KUKA KRL program: ps_ltc_geo_x1.src, ps_ltc_geo_x1.dat

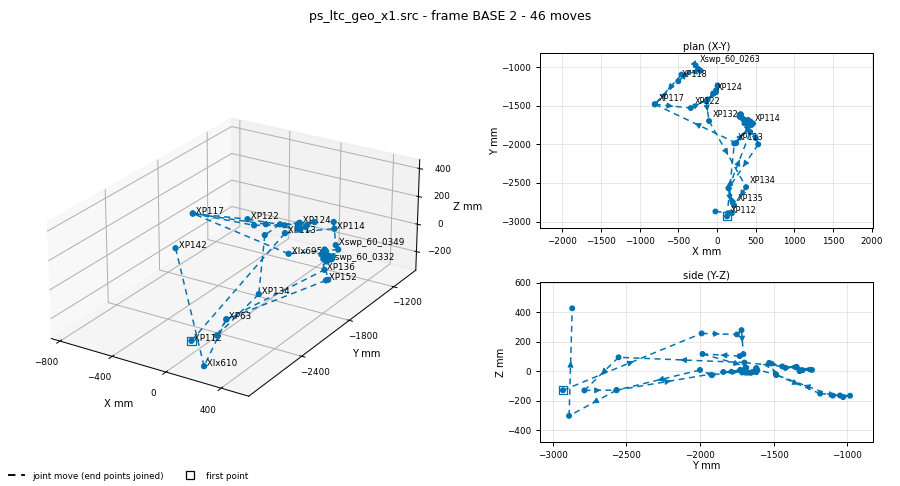
[picture p0: tool path of ps_ltc_geo_x1.src in frame BASE 2, 46 of 48 moves have a stored position in this frame; points joined in program order, loops and branches not executed]
--- ps_ltc_geo_x1.src ---
&ACCESS RVO2
&REL 17
&COMMENT Solda GUN X1 geometria
&PARAM DISKPATH = KRC:\R1\Program\SOLDA LTC
DEF ps_ltc_geo_x1( )
;FOLD INI
  ;FOLD BASISTECH INI
    GLOBAL INTERRUPT DECL 3 WHEN $STOPMESS==TRUE DO IR_STOPM ( )
    INTERRUPT ON 3
    BAS (#INITMOV,0 )
  ;ENDFOLD (BASISTECH INI)
;FOLD SPOTTECH INI
USERSPOT(#INIT)
;ENDFOLD (SPOTTECH INI)
;FOLD GRIPPERTECH INI
USER_GRP(0,DUMMY,DUMMY,GDEFAULT)
;ENDFOLD (GRIPPERTECH INI)
  ;FOLD USER INI
    ;Make your modifications here

  ;ENDFOLD (USER INI)
;ENDFOLD (INI)

; Caracterização dos meios de produção:
; Versão Atual:
; 08/06/2013 12:00 Name: P13.050-R1 CHANGES: Solda Geometria Accelo
; Gun X1 (F2 6640 0018 985)

chk_w1_wechs_ok ( )              ; CHECK X1

if MaxStandMenge (4) then
 MaxStandmengeErreicht (4)
endif

IF (NOT(GHOST())) THEN
if Elektrodenwechsel (4) then
 e_fraes1 ()
endif
ENDIF

;FOLD PTP P112 Vel=100 % PDAT114 Tool[1]:GUN X1 Base[2]:Accelo;%{PE}%R 8.2.20,%MKUKATPBASIS,%CMOVE,%VPTP,%P 1:PTP, 2:P112, 3:, 5:100, 7:PDAT114
$BWDSTART=FALSE
PDAT_ACT=PPDAT114
FDAT_ACT=FP112
BAS(#PTP_PARAMS,100)
PTP XP112
;ENDFOLD

;FOLD OUT 3339 'R1 solicita lib soldar geometria' State=TRUE ;%{PE}%R 8.2.20,%MKUKATPBASIS,%COUT,%VOUTX,%P 2:3339, 3:R1 solicita lib soldar geometria, 5:TRUE, 6:
$OUT[3339]=TRUE
;ENDFOLD
;FOLD WAIT FOR ( IN 3339 'Aguarda lib. Soldar geometria' );%{PE}%R 8.2.20,%MKUKATPBASIS,%CEXT_WAIT_FOR,%VEXT_WAIT_FOR,%P 2:, 4:, 5:$IN, 6:3339, 7:Aguarda lib. Soldar geometria, 9:
WAIT FOR  ( $IN[3339] )
;ENDFOLD
;FOLD OUT 3339 'R1 solicita lib soldar geometria' State=FALSE ;%{PE}%R 8.2.20,%MKUKATPBASIS,%COUT,%VOUTX,%P 2:3339, 3:R1 solicita lib soldar geometria, 5:FALSE, 6:
$OUT[3339]=FALSE
;ENDFOLD
;FOLD OUT 3348 'Fora area GEOBOX' State=FALSE ;%{PE}%R 8.2.20,%MKUKATPBASIS,%COUT,%VOUTX,%P 2:3348, 3:Fora area GEOBOX, 5:FALSE, 6:
$OUT[3348]=FALSE
;ENDFOLD

;FOLD Collision.Monitoring_3_On ;%{PE}%MKUKATPUSER
COLLSTOP( 3, 1 ) ;Interrupt-Controlled
;ENDFOLD
;FOLD Collision.Monitoring_AREA_1_On ;%{PE}%MKUKATPUSER
COLLSTOP( 7, 1 ) ;not Interrupt-Controlled
;ENDFOLD

;FOLD PTP P113 CONT Vel=100 % PDAT115 Tool[1]:GUN X1 Base[2]:Accelo;%{PE}%R 8.2.20,%MKUKATPBASIS,%CMOVE,%VPTP,%P 1:PTP, 2:P113, 3:C_DIS, 5:100, 7:PDAT115
$BWDSTART=FALSE
PDAT_ACT=PPDAT115
FDAT_ACT=FP113
BAS(#PTP_PARAMS,100)
PTP XP113 C_DIS
;ENDFOLD
;FOLD PTP P114 CONT Vel=100 % PDAT116 Tool[1]:GUN X1 Base[2]:Accelo;%{PE}%R 8.2.20,%MKUKATPBASIS,%CMOVE,%VPTP,%P 1:PTP, 2:P114, 3:C_DIS, 5:100, 7:PDAT116
$BWDSTART=FALSE
PDAT_ACT=PPDAT116
FDAT_ACT=FP114
BAS(#PTP_PARAMS,100)
PTP XP114 C_DIS
;ENDFOLD

;FOLD ; swp_60_0355;%{PE}%R 8.2.20,%MKUKATPBASIS,%CCOMMENT,%VNORMAL,%P 2:swp_60_0355
;ENDFOLD
;FOLD PTP swp_60_0355 P_OLP80 SPOT Gun=4 RETR CLS PGNO1=106 ACTIVE=1 Tool[1]:GUN X1 Base[2]:Accelo;%{PE}%R 8.2.2,%MKUKATPSPOT,%CSPOT,%VPTP,%P 1:PTP, 2:swp_60_0355, 3:, 5:100, 7:P_OLP80, 10:4, 12:#FIRST, 14:#CLO, 16:187, 18:1, 20:1, 22:0, 24:1, 25:S_OLP4
$BWDSTART=FALSE
PDAT_ACT=PP_OLP80
FDAT_ACT=Fswp_60_0355
BAS(#PTP_PARAMS,PP_OLP80.VEL)
S_ACT.GUN=4
S_ACT.PAIR=SDEFAULT.PAIR
S_ACT.RETR=#CLO
S_ACT.CLO_TM=1
S_ACT.PGNO1=106
S_ACT.PGNO2=SDEFAULT.PGNO2
S_ACT.PRESS1=SDEFAULT.PRESS1
S_ACT.PRESS2=SDEFAULT.PRESS2
S_READY=FALSE
PTP Xswp_60_0355
USERSPOT(#SPOT, S_ACT)
WAIT FOR S_READY
;ENDFOLD

;FOLD ; swp_60_0349;%{PE}%R 8.2.20,%MKUKATPBASIS,%CCOMMENT,%VNORMAL,%P 2:swp_60_0349
;ENDFOLD
;FOLD PTP swp_60_0349 P_OLP81 SPOT Gun=4 RETR OPN PGNO1=105 ACTIVE=1 Tool[1]:GUN X1 Base[2]:Accelo;%{PE}%R 8.2.2,%MKUKATPSPOT,%CSPOT,%VPTP,%P 1:PTP, 2:swp_60_0349, 3:, 5:100, 7:P_OLP81, 10:4, 12:#FIRST, 14:#OPN, 16:186, 18:1, 20:1, 22:0, 24:1, 25:S_OLP5
$BWDSTART=FALSE
PDAT_ACT=PP_OLP81
FDAT_ACT=Fswp_60_0349
BAS(#PTP_PARAMS,PP_OLP81.VEL)
S_ACT.GUN=4
S_ACT.PAIR=SDEFAULT.PAIR
S_ACT.RETR=#OPN
S_ACT.CLO_TM=1
S_ACT.PGNO1=105
S_ACT.PGNO2=SDEFAULT.PGNO2
S_ACT.PRESS1=SDEFAULT.PRESS1
S_ACT.PRESS2=SDEFAULT.PRESS2
S_READY=FALSE
PTP Xswp_60_0349
USERSPOT(#SPOT, S_ACT)
WAIT FOR S_READY
;ENDFOLD

;FOLD PTP P115 CONT Vel=100 % PDAT117 Tool[1]:GUN X1 Base[2]:Accelo;%{PE}%R 8.2.20,%MKUKATPBASIS,%CMOVE,%VPTP,%P 1:PTP, 2:P115, 3:C_DIS, 5:100, 7:PDAT117
$BWDSTART=FALSE
PDAT_ACT=PPDAT117
FDAT_ACT=FP115
BAS(#PTP_PARAMS,100)
PTP XP115 C_DIS
;ENDFOLD
;FOLD PTP lx695 Vel=100 % P_OLP82 Tool[1]:GUN X1 Base[2]:Accelo;%{PE}%R 8.2.20,%MKUKATPBASIS,%CMOVE,%VPTP,%P 1:PTP, 2:lx695, 3:, 5:100, 7:P_OLP82
$BWDSTART=FALSE
PDAT_ACT=PP_OLP82
FDAT_ACT=Flx695
BAS(#PTP_PARAMS,100)
PTP Xlx695
;ENDFOLD

;FOLD Collision.Monitoring_AREA_3_On ;%{PE}%MKUKATPUSER
COLLSTOP( 9, 1 ) ;not Interrupt-Controlled
;ENDFOLD

;FOLD PTP P117 CONT Vel=100 % PDAT119 Tool[1]:GUN X1 Base[2]:Accelo;%{PE}%R 8.2.20,%MKUKATPBASIS,%CMOVE,%VPTP,%P 1:PTP, 2:P117, 3:C_DIS, 5:100, 7:PDAT119
$BWDSTART=FALSE
PDAT_ACT=PPDAT119
FDAT_ACT=FP117
BAS(#PTP_PARAMS,100)
PTP XP117 C_DIS
;ENDFOLD
;FOLD PTP P118 CONT Vel=100 % PDAT120 Tool[1]:GUN X1 Base[2]:Accelo;%{PE}%R 8.2.20,%MKUKATPBASIS,%CMOVE,%VPTP,%P 1:PTP, 2:P118, 3:C_DIS, 5:100, 7:PDAT120
$BWDSTART=FALSE
PDAT_ACT=PPDAT120
FDAT_ACT=FP118
BAS(#PTP_PARAMS,100)
PTP XP118 C_DIS
;ENDFOLD

;FOLD ; swp_60_0263;%{PE}%R 8.2.20,%MKUKATPBASIS,%CCOMMENT,%VNORMAL,%P 2:swp_60_0263
;ENDFOLD
;FOLD PTP swp_60_0263 PDAT121 SPOT Gun=4 RETR CLS PGNO1=100 ACTIVE=1 Tool[1]:GUN X1 Base[2]:Accelo;%{PE}%R 8.2.2,%MKUKATPSPOT,%CSPOT,%VPTP,%P 1:PTP, 2:swp_60_0263, 3:, 5:100, 7:PDAT121, 10:4, 12:#FIRST, 14:#CLO, 16:181, 18:1, 20:0, 22:0, 24:1, 25:NORMAL
$BWDSTART=FALSE
PDAT_ACT=PPDAT121
FDAT_ACT=Fswp_60_0263
BAS(#PTP_PARAMS,PPDAT121.VEL)
S_ACT.GUN=4
S_ACT.PAIR=SDEFAULT.PAIR
S_ACT.RETR=#CLO
S_ACT.CLO_TM=1
S_ACT.PGNO1=100
S_ACT.PGNO2=SDEFAULT.PGNO2
S_ACT.PRESS1=SDEFAULT.PRESS1
S_ACT.PRESS2=SDEFAULT.PRESS2
S_READY=FALSE
PTP Xswp_60_0263
USERSPOT(#SPOT, S_ACT)
WAIT FOR S_READY
;ENDFOLD

;FOLD PTP P120 CONT Vel=100 % PDAT122 Tool[1]:GUN X1 Base[2]:Accelo;%{PE}%R 8.2.20,%MKUKATPBASIS,%CMOVE,%VPTP,%P 1:PTP, 2:P120, 3:C_DIS, 5:100, 7:PDAT122
$BWDSTART=FALSE
PDAT_ACT=PPDAT122
FDAT_ACT=FP120
BAS(#PTP_PARAMS,100)
PTP XP120 C_DIS
;ENDFOLD

;FOLD ; 60_0267;%{PE}%R 8.2.20,%MKUKATPBASIS,%CCOMMENT,%VNORMAL,%P 2:60_0267
;ENDFOLD
;FOLD PTP swp_60_0267 PDAT123 SPOT Gun=4 RETR OPN PGNO1=101 ACTIVE=1 Tool[1]:GUN X1 Base[2]:Accelo;%{PE}%R 8.2.2,%MKUKATPSPOT,%CSPOT,%VPTP,%P 1:PTP, 2:swp_60_0267, 3:, 5:100, 7:PDAT123, 10:4, 12:#FIRST, 14:#OPN, 16:182, 18:1, 20:0, 22:0, 24:1, 25:NORMAL
$BWDSTART=FALSE
PDAT_ACT=PPDAT123
FDAT_ACT=Fswp_60_0267
BAS(#PTP_PARAMS,PPDAT123.VEL)
S_ACT.GUN=4
S_ACT.PAIR=SDEFAULT.PAIR
S_ACT.RETR=#OPN
S_ACT.CLO_TM=1
S_ACT.PGNO1=101
S_ACT.PGNO2=SDEFAULT.PGNO2
S_ACT.PRESS1=SDEFAULT.PRESS1
S_ACT.PRESS2=SDEFAULT.PRESS2
S_READY=FALSE
PTP Xswp_60_0267
USERSPOT(#SPOT, S_ACT)
WAIT FOR S_READY
;ENDFOLD

;FOLD PTP lx696 CONT Vel=100 % P_OLP83 Tool[1]:GUN X1 Base[2]:Accelo;%{PE}%R 8.2.20,%MKUKATPBASIS,%CMOVE,%VPTP,%P 1:PTP, 2:lx696, 3:C_DIS, 5:100, 7:P_OLP83
$BWDSTART=FALSE
PDAT_ACT=PP_OLP83
FDAT_ACT=Flx696
BAS(#PTP_PARAMS,100)
PTP Xlx696 C_DIS
;ENDFOLD
;FOLD PTP lx697 CONT Vel=100 % P_OLP84 Tool[1]:GUN X1 Base[2]:Accelo;%{PE}%R 8.2.20,%MKUKATPBASIS,%CMOVE,%VPTP,%P 1:PTP, 2:lx697, 3:C_DIS, 5:100, 7:P_OLP84
$BWDSTART=FALSE
PDAT_ACT=PP_OLP84
FDAT_ACT=Flx697
BAS(#PTP_PARAMS,100)
PTP Xlx697 C_DIS
;ENDFOLD

;FOLD PTP P122 CONT Vel=100 % PDAT124 Tool[1]:GUN X1 Base[2]:Accelo;%{PE}%R 8.2.20,%MKUKATPBASIS,%CMOVE,%VPTP,%P 1:PTP, 2:P122, 3:C_DIS, 5:100, 7:PDAT124
$BWDSTART=FALSE
PDAT_ACT=PPDAT124
FDAT_ACT=FP122
BAS(#PTP_PARAMS,100)
PTP XP122 C_DIS
;ENDFOLD
;FOLD PTP P123 CONT Vel=100 % PDAT125 Tool[1]:GUN X1 Base[2]:Accelo;%{PE}%R 8.2.20,%MKUKATPBASIS,%CMOVE,%VPTP,%P 1:PTP, 2:P123, 3:C_DIS, 5:100, 7:PDAT125
$BWDSTART=FALSE
PDAT_ACT=PPDAT125
FDAT_ACT=FP123
BAS(#PTP_PARAMS,100)
PTP XP123 C_DIS
;ENDFOLD
;FOLD PTP P124 CONT Vel=100 % PDAT126 Tool[1]:GUN X1 Base[2]:Accelo;%{PE}%R 8.2.20,%MKUKATPBASIS,%CMOVE,%VPTP,%P 1:PTP, 2:P124, 3:C_DIS, 5:100, 7:PDAT126
$BWDSTART=FALSE
PDAT_ACT=PPDAT126
FDAT_ACT=FP124
BAS(#PTP_PARAMS,100)
PTP XP124 C_DIS
;ENDFOLD
;FOLD PTP P147 CONT Vel=100 % PDAT154 Tool[1]:GUN X1 Base[2]:Accelo;%{PE}%R 8.2.20,%MKUKATPBASIS,%CMOVE,%VPTP,%P 1:PTP, 2:P147, 3:C_DIS, 5:100, 7:PDAT154
$BWDSTART=FALSE
PDAT_ACT=PPDAT154
FDAT_ACT=FP147
BAS(#PTP_PARAMS,100)
PTP XP147 C_DIS
;ENDFOLD
;FOLD PTP P125 CONT Vel=100 % PDAT127 Tool[1]:GUN X1 Base[2]:Accelo;%{PE}%R 8.2.20,%MKUKATPBASIS,%CMOVE,%VPTP,%P 1:PTP, 2:P125, 3:C_DIS, 5:100, 7:PDAT127
$BWDSTART=FALSE
PDAT_ACT=PPDAT127
FDAT_ACT=FP125
BAS(#PTP_PARAMS,100)
PTP XP125 C_DIS
;ENDFOLD

;FOLD ; swp_60_0283;%{PE}%R 8.2.20,%MKUKATPBASIS,%CCOMMENT,%VNORMAL,%P 2:swp_60_0283
;ENDFOLD
;FOLD PTP swp_60_0283 P_OLP85 SPOT Gun=4 RETR OPN PGNO1=102 ACTIVE=1 Tool[1]:GUN X1 Base[2]:Accelo;%{PE}%R 8.2.2,%MKUKATPSPOT,%CSPOT,%VPTP,%P 1:PTP, 2:swp_60_0283, 3:, 5:100, 7:P_OLP85, 10:4, 12:#FIRST, 14:#OPN, 16:183, 18:1, 20:1, 22:0, 24:1, 25:S_OLP3
$BWDSTART=FALSE
PDAT_ACT=PP_OLP85
FDAT_ACT=Fswp_60_0283
BAS(#PTP_PARAMS,PP_OLP85.VEL)
S_ACT.GUN=4
S_ACT.PAIR=SDEFAULT.PAIR
S_ACT.RETR=#OPN
S_ACT.CLO_TM=1
S_ACT.PGNO1=102
S_ACT.PGNO2=SDEFAULT.PGNO2
S_ACT.PRESS1=SDEFAULT.PRESS1
S_ACT.PRESS2=SDEFAULT.PRESS2
S_READY=FALSE
PTP Xswp_60_0283
USERSPOT(#SPOT, S_ACT)
WAIT FOR S_READY
;ENDFOLD

;FOLD PTP P126 CONT Vel=100 % PDAT128 Tool[1]:GUN X1 Base[2]:Accelo;%{PE}%R 8.2.20,%MKUKATPBASIS,%CMOVE,%VPTP,%P 1:PTP, 2:P126, 3:C_DIS, 5:100, 7:PDAT128
$BWDSTART=FALSE
PDAT_ACT=PPDAT128
FDAT_ACT=FP126
BAS(#PTP_PARAMS,100)
PTP XP126 C_DIS
;ENDFOLD
;FOLD PTP P127 CONT Vel=100 % PDAT129 Tool[1]:GUN X1 Base[2]:Accelo;%{PE}%R 8.2.20,%MKUKATPBASIS,%CMOVE,%VPTP,%P 1:PTP, 2:P127, 3:C_DIS, 5:100, 7:PDAT129
$BWDSTART=FALSE
PDAT_ACT=PPDAT129
FDAT_ACT=FP127
BAS(#PTP_PARAMS,100)
PTP XP127 C_DIS
;ENDFOLD
;FOLD PTP P132 CONT Vel=100 % PDAT134 Tool[1]:GUN X1 Base[2]:Accelo;%{PE}%R 8.2.20,%MKUKATPBASIS,%CMOVE,%VPTP,%P 1:PTP, 2:P132, 3:C_DIS, 5:100, 7:PDAT134
$BWDSTART=FALSE
PDAT_ACT=PPDAT134
FDAT_ACT=FP132
BAS(#PTP_PARAMS,100)
PTP XP132 C_DIS
;ENDFOLD
;FOLD PTP P134 CONT Vel=100 % PDAT136 Tool[1]:GUN X1 Base[2]:Accelo;%{PE}%R 8.2.20,%MKUKATPBASIS,%CMOVE,%VPTP,%P 1:PTP, 2:P134, 3:C_DIS, 5:100, 7:PDAT136
$BWDSTART=FALSE
PDAT_ACT=PPDAT136
FDAT_ACT=FP134
BAS(#PTP_PARAMS,100)
PTP XP134 C_DIS
;ENDFOLD

;FOLD Collision.Monitoring_AREA_1_Off . ;%{PE}%MKUKATPUSER
COLLSTOP( 7, 2+0 )
;ENDFOLD
;FOLD Collision.Monitoring_AREA_3_Off . ;%{PE}%MKUKATPUSER
COLLSTOP( 9, 2+0 )
;ENDFOLD
;FOLD Collision.Monitoring_AREA_5_Off . ;%{PE}%MKUKATPUSER
COLLSTOP( 11, 2+0 )
;ENDFOLD
;FOLD Collision.Monitoring_3_Off . ;%{PE}%MKUKATPUSER
COLLSTOP( 3, 2+0 )
;ENDFOLD

;FOLD PTP P135 CONT Vel=100 % PDAT137 Tool[1]:GUN X1 Base[2]:Accelo;%{PE}%R 8.2.20,%MKUKATPBASIS,%CMOVE,%VPTP,%P 1:PTP, 2:P135, 3:C_DIS, 5:100, 7:PDAT137
$BWDSTART=FALSE
PDAT_ACT=PPDAT137
FDAT_ACT=FP135
BAS(#PTP_PARAMS,100)
PTP XP135 C_DIS
;ENDFOLD
;FOLD PTP P63 CONT Vel=100 % PDAT65 Tool[1]:GUN X1 Base[2]:Accelo;%{PE}%R 8.2.20,%MKUKATPBASIS,%CMOVE,%VPTP,%P 1:PTP, 2:P63, 3:C_DIS, 5:100, 7:PDAT65
$BWDSTART=FALSE
PDAT_ACT=PPDAT65
FDAT_ACT=FP63
BAS(#PTP_PARAMS,100)
PTP XP63 C_DIS
;ENDFOLD
;FOLD PTP P136 CONT Vel=100 % PDAT138 Tool[1]:GUN X1 Base[2]:Accelo;%{PE}%R 8.2.20,%MKUKATPBASIS,%CMOVE,%VPTP,%P 1:PTP, 2:P136, 3:C_DIS, 5:100, 7:PDAT138
$BWDSTART=FALSE
PDAT_ACT=PPDAT138
FDAT_ACT=FP136
BAS(#PTP_PARAMS,100)
PTP XP136 C_DIS
;ENDFOLD

;FOLD Collision.Monitoring_AREA_4_On ;%{PE}%MKUKATPUSER
COLLSTOP( 10, 1 ) ;not Interrupt-Controlled
;ENDFOLD

;FOLD PTP lx698 CONT Vel=100 % P_OLP88 Tool[1]:GUN X1 Base[2]:Accelo;%{PE}%R 8.2.20,%MKUKATPBASIS,%CMOVE,%VPTP,%P 1:PTP, 2:lx698, 3:C_DIS, 5:100, 7:P_OLP88
$BWDSTART=FALSE
PDAT_ACT=PP_OLP88
FDAT_ACT=Flx698
BAS(#PTP_PARAMS,100)
PTP Xlx698 C_DIS
;ENDFOLD

end_weld_geo()         ; Bit fim geometria
;FOLD OUT 3331 'SOLDANDO Respot 7 pontos' State=TRUE ;%{PE}%R 8.2.20,%MKUKATPBASIS,%COUT,%VOUTX,%P 2:3331, 3:SOLDANDO Respot 7 pontos, 5:TRUE, 6:
$OUT[3331]=TRUE
;ENDFOLD
;FOLD WAIT FOR ( IN 3332 'LIBERA Respot' );%{PE}%R 8.2.20,%MKUKATPBASIS,%CEXT_WAIT_FOR,%VEXT_WAIT_FOR,%P 2:, 4:, 5:$IN, 6:3332, 7:LIBERA Respot, 9:
WAIT FOR  ( $IN[3332] )
;ENDFOLD

;FOLD PTP P143 CONT Vel=100 % PDAT150 Tool[1]:GUN X1 Base[2]:Accelo;%{PE}%R 8.2.20,%MKUKATPBASIS,%CMOVE,%VPTP,%P 1:PTP, 2:P143, 3:C_DIS, 5:100, 7:PDAT150
$BWDSTART=FALSE
PDAT_ACT=PPDAT150
FDAT_ACT=FP143
BAS(#PTP_PARAMS,100)
PTP XP143 C_DIS
;ENDFOLD

;FOLD ; swp_60_0315;%{PE}%R 8.2.20,%MKUKATPBASIS,%CCOMMENT,%VNORMAL,%P 2:swp_60_0315
;ENDFOLD
;FOLD PTP swp_60_0315 PDAT149 SPOT Gun=4 RETR CLS PGNO1=132 ACTIVE=1 Tool[1]:GUN X1 Base[0];%{PE}%R 8.2.2,%MKUKATPSPOT,%CSPOT,%VPTP,%P 1:PTP, 2:swp_60_0315, 3:, 5:100, 7:PDAT149, 10:4, 12:#FIRST, 14:#CLO, 16:213, 18:1, 20:0, 22:0, 24:1, 25:NORMAL
$BWDSTART=FALSE
PDAT_ACT=PPDAT149
FDAT_ACT=Fswp_60_0315
BAS(#PTP_PARAMS,PPDAT149.VEL)
S_ACT.GUN=4
S_ACT.PAIR=SDEFAULT.PAIR
S_ACT.RETR=#CLO
S_ACT.CLO_TM=1
S_ACT.PGNO1=132
S_ACT.PGNO2=SDEFAULT.PGNO2
S_ACT.PRESS1=SDEFAULT.PRESS1
S_ACT.PRESS2=SDEFAULT.PRESS2
S_READY=FALSE
PTP Xswp_60_0315
USERSPOT(#SPOT, S_ACT)
WAIT FOR S_READY
;ENDFOLD

;FOLD PTP P144 CONT Vel=100 % PDAT151 Tool[1]:GUN X1 Base[2]:Accelo;%{PE}%R 8.2.20,%MKUKATPBASIS,%CMOVE,%VPTP,%P 1:PTP, 2:P144, 3:C_DIS, 5:100, 7:PDAT151
$BWDSTART=FALSE
PDAT_ACT=PPDAT151
FDAT_ACT=FP144
BAS(#PTP_PARAMS,100)
PTP XP144 C_DIS
;ENDFOLD

;FOLD ; swp_60_0317;%{PE}%R 8.2.20,%MKUKATPBASIS,%CCOMMENT,%VNORMAL,%P 2:swp_60_0317
;ENDFOLD
;FOLD PTP swp_60_0317 P_OLP89 SPOT Gun=4 RETR CLS PGNO1=107 ACTIVE=1 Tool[1]:GUN X1 Base[2]:Accelo;%{PE}%R 8.2.2,%MKUKATPSPOT,%CSPOT,%VPTP,%P 1:PTP, 2:swp_60_0317, 3:, 5:100, 7:P_OLP89, 10:4, 12:#FIRST, 14:#CLO, 16:188, 18:1, 20:1, 22:0, 24:1, 25:S_OLP3
$BWDSTART=FALSE
PDAT_ACT=PP_OLP89
FDAT_ACT=Fswp_60_0317
BAS(#PTP_PARAMS,PP_OLP89.VEL)
S_ACT.GUN=4
S_ACT.PAIR=SDEFAULT.PAIR
S_ACT.RETR=#CLO
S_ACT.CLO_TM=1
S_ACT.PGNO1=107
S_ACT.PGNO2=SDEFAULT.PGNO2
S_ACT.PRESS1=SDEFAULT.PRESS1
S_ACT.PRESS2=SDEFAULT.PRESS2
S_READY=FALSE
PTP Xswp_60_0317
USERSPOT(#SPOT, S_ACT)
WAIT FOR S_READY
;ENDFOLD

;FOLD PTP P145 CONT Vel=100 % PDAT152 Tool[1]:GUN X1 Base[2]:Accelo;%{PE}%R 8.2.20,%MKUKATPBASIS,%CMOVE,%VPTP,%P 1:PTP, 2:P145, 3:C_DIS, 5:100, 7:PDAT152
$BWDSTART=FALSE
PDAT_ACT=PPDAT152
FDAT_ACT=FP145
BAS(#PTP_PARAMS,100)
PTP XP145 C_DIS
;ENDFOLD

;FOLD ; swp_60_0319;%{PE}%R 8.2.20,%MKUKATPBASIS,%CCOMMENT,%VNORMAL,%P 2:swp_60_0319
;ENDFOLD
;FOLD PTP swp_60_0331 PDAT155 SPOT Gun=4 RETR CLS PGNO1=133 ACTIVE=1 Tool[1]:GUN X1 Base[2]:Accelo;%{PE}%R 8.2.2,%MKUKATPSPOT,%CSPOT,%VPTP,%P 1:PTP, 2:swp_60_0331, 3:, 5:100, 7:PDAT155, 10:4, 12:#FIRST, 14:#CLO, 16:214, 18:1, 20:0, 22:0, 24:1, 25:NORMAL
$BWDSTART=FALSE
PDAT_ACT=PPDAT155
FDAT_ACT=Fswp_60_0331
BAS(#PTP_PARAMS,PPDAT155.VEL)
S_ACT.GUN=4
S_ACT.PAIR=SDEFAULT.PAIR
S_ACT.RETR=#CLO
S_ACT.CLO_TM=1
S_ACT.PGNO1=133
S_ACT.PGNO2=SDEFAULT.PGNO2
S_ACT.PRESS1=SDEFAULT.PRESS1
S_ACT.PRESS2=SDEFAULT.PRESS2
S_READY=FALSE
PTP Xswp_60_0331
USERSPOT(#SPOT, S_ACT)
WAIT FOR S_READY
;ENDFOLD

;FOLD ; swp_60_0321;%{PE}%R 8.2.20,%MKUKATPBASIS,%CCOMMENT,%VNORMAL,%P 2:swp_60_0321
;ENDFOLD
;FOLD PTP swp_60_0321 PDAT139 SPOT Gun=4 RETR CLS PGNO1=134 ACTIVE=1 Tool[1]:GUN X1 Base[2]:Accelo;%{PE}%R 8.2.2,%MKUKATPSPOT,%CSPOT,%VPTP,%P 1:PTP, 2:swp_60_0321, 3:, 5:100, 7:PDAT139, 10:4, 12:#FIRST, 14:#CLO, 16:215, 18:1, 20:0, 22:0, 24:1, 25:NORMAL
$BWDSTART=FALSE
PDAT_ACT=PPDAT139
FDAT_ACT=Fswp_60_0321
BAS(#PTP_PARAMS,PPDAT139.VEL)
S_ACT.GUN=4
S_ACT.PAIR=SDEFAULT.PAIR
S_ACT.RETR=#CLO
S_ACT.CLO_TM=1
S_ACT.PGNO1=134
S_ACT.PGNO2=SDEFAULT.PGNO2
S_ACT.PRESS1=SDEFAULT.PRESS1
S_ACT.PRESS2=SDEFAULT.PRESS2
S_READY=FALSE
PTP Xswp_60_0321
USERSPOT(#SPOT, S_ACT)
WAIT FOR S_READY
;ENDFOLD

;FOLD ; swp_60_0323;%{PE}%R 8.2.20,%MKUKATPBASIS,%CCOMMENT,%VNORMAL,%P 2:swp_60_0323
;ENDFOLD
;FOLD PTP swp_60_0332 PDAT156 SPOT Gun=4 RETR CLS PGNO1=135 ACTIVE=1 Tool[1]:GUN X1 Base[2]:Accelo;%{PE}%R 8.2.2,%MKUKATPSPOT,%CSPOT,%VPTP,%P 1:PTP, 2:swp_60_0332, 3:, 5:100, 7:PDAT156, 10:4, 12:#FIRST, 14:#CLO, 16:216, 18:1, 20:0, 22:0, 24:1, 25:NORMAL
$BWDSTART=FALSE
PDAT_ACT=PPDAT156
FDAT_ACT=Fswp_60_0332
BAS(#PTP_PARAMS,PPDAT156.VEL)
S_ACT.GUN=4
S_ACT.PAIR=SDEFAULT.PAIR
S_ACT.RETR=#CLO
S_ACT.CLO_TM=1
S_ACT.PGNO1=135
S_ACT.PGNO2=SDEFAULT.PGNO2
S_ACT.PRESS1=SDEFAULT.PRESS1
S_ACT.PRESS2=SDEFAULT.PRESS2
S_READY=FALSE
PTP Xswp_60_0332
USERSPOT(#SPOT, S_ACT)
WAIT FOR S_READY
;ENDFOLD

;FOLD PTP P148 CONT Vel=100 % PDAT157 Tool[1]:GUN X1 Base[2]:Accelo;%{PE}%R 8.2.20,%MKUKATPBASIS,%CMOVE,%VPTP,%P 1:PTP, 2:P148, 3:C_DIS, 5:100, 7:PDAT157
$BWDSTART=FALSE
PDAT_ACT=PPDAT157
FDAT_ACT=FP148
BAS(#PTP_PARAMS,100)
PTP XP148 C_DIS
;ENDFOLD
;FOLD PTP P149 CONT Vel=100 % PDAT158 Tool[1]:GUN X1 Base[2]:Accelo;%{PE}%R 8.2.20,%MKUKATPBASIS,%CMOVE,%VPTP,%P 1:PTP, 2:P149, 3:C_DIS, 5:100, 7:PDAT158
$BWDSTART=FALSE
PDAT_ACT=PPDAT158
FDAT_ACT=FP149
BAS(#PTP_PARAMS,100)
PTP XP149 C_DIS
;ENDFOLD

;FOLD ; swp_60_0325;%{PE}%R 8.2.20,%MKUKATPBASIS,%CCOMMENT,%VNORMAL,%P 2:swp_60_0325
;ENDFOLD
;FOLD PTP swp_60_0325 PDAT140 SPOT Gun=4 RETR CLS PGNO1=109 ACTIVE=1 Tool[1]:GUN X1 Base[2]:Accelo;%{PE}%R 8.2.2,%MKUKATPSPOT,%CSPOT,%VPTP,%P 1:PTP, 2:swp_60_0325, 3:, 5:100, 7:PDAT140, 10:4, 12:#FIRST, 14:#CLO, 16:190, 18:1, 20:0, 22:0, 24:1, 25:NORMAL
$BWDSTART=FALSE
PDAT_ACT=PPDAT140
FDAT_ACT=Fswp_60_0325
BAS(#PTP_PARAMS,PPDAT140.VEL)
S_ACT.GUN=4
S_ACT.PAIR=SDEFAULT.PAIR
S_ACT.RETR=#CLO
S_ACT.CLO_TM=1
S_ACT.PGNO1=109
S_ACT.PGNO2=SDEFAULT.PGNO2
S_ACT.PRESS1=SDEFAULT.PRESS1
S_ACT.PRESS2=SDEFAULT.PRESS2
S_READY=FALSE
PTP Xswp_60_0325
USERSPOT(#SPOT, S_ACT)
WAIT FOR S_READY
;ENDFOLD

;FOLD Collision.Monitoring_3_Off . ;%{PE}%MKUKATPUSER
COLLSTOP( 3, 2+0 )
;ENDFOLD

;FOLD PTP P146 CONT Vel=100 % PDAT153 Tool[1]:GUN X1 Base[2]:Accelo;%{PE}%R 8.2.20,%MKUKATPBASIS,%CMOVE,%VPTP,%P 1:PTP, 2:P146, 3:C_DIS, 5:100, 7:PDAT153
$BWDSTART=FALSE
PDAT_ACT=PPDAT153
FDAT_ACT=FP146
BAS(#PTP_PARAMS,100)
PTP XP146 C_DIS
;ENDFOLD

;FOLD ; swp_60_0327;%{PE}%R 8.2.20,%MKUKATPBASIS,%CCOMMENT,%VNORMAL,%P 2:swp_60_0327
;ENDFOLD
;FOLD PTP swp_60_0327 PDAT141 SPOT Gun=4 RETR OPN PGNO1=136 ACTIVE=1 Tool[1]:GUN X1 Base[0];%{PE}%R 8.2.2,%MKUKATPSPOT,%CSPOT,%VPTP,%P 1:PTP, 2:swp_60_0327, 3:, 5:100, 7:PDAT141, 10:4, 12:#FIRST, 14:#OPN, 16:217, 18:1, 20:0, 22:0, 24:1, 25:NORMAL
$BWDSTART=FALSE
PDAT_ACT=PPDAT141
FDAT_ACT=Fswp_60_0327
BAS(#PTP_PARAMS,PPDAT141.VEL)
S_ACT.GUN=4
S_ACT.PAIR=SDEFAULT.PAIR
S_ACT.RETR=#OPN
S_ACT.CLO_TM=1
S_ACT.PGNO1=136
S_ACT.PGNO2=SDEFAULT.PGNO2
S_ACT.PRESS1=SDEFAULT.PRESS1
S_ACT.PRESS2=SDEFAULT.PRESS2
S_READY=FALSE
PTP Xswp_60_0327
USERSPOT(#SPOT, S_ACT)
WAIT FOR S_READY
;ENDFOLD

;FOLD PTP P150 CONT Vel=100 % PDAT159 Tool[1]:GUN X1 Base[2]:Accelo;%{PE}%R 8.2.20,%MKUKATPBASIS,%CMOVE,%VPTP,%P 1:PTP, 2:P150, 3:C_DIS, 5:100, 7:PDAT159
$BWDSTART=FALSE
PDAT_ACT=PPDAT159
FDAT_ACT=FP150
BAS(#PTP_PARAMS,100)
PTP XP150 C_DIS
;ENDFOLD
;FOLD PTP P151 Vel=100 % PDAT160 Tool[1]:GUN X1 Base[2]:Accelo;%{PE}%R 8.2.20,%MKUKATPBASIS,%CMOVE,%VPTP,%P 1:PTP, 2:P151, 3:, 5:100, 7:PDAT160
$BWDSTART=FALSE
PDAT_ACT=PPDAT160
FDAT_ACT=FP151
BAS(#PTP_PARAMS,100)
PTP XP151
;ENDFOLD

;FOLD Collision.Monitoring_AREA_4_Off . ;%{PE}%MKUKATPUSER
COLLSTOP( 10, 2+0 )
;ENDFOLD

;FOLD PTP P140 CONT Vel=100 % PDAT146 Tool[1]:GUN X1 Base[2]:Accelo;%{PE}%R 8.2.20,%MKUKATPBASIS,%CMOVE,%VPTP,%P 1:PTP, 2:P140, 3:C_DIS, 5:100, 7:PDAT146
$BWDSTART=FALSE
PDAT_ACT=PPDAT146
FDAT_ACT=FP140
BAS(#PTP_PARAMS,100)
PTP XP140 C_DIS
;ENDFOLD
;FOLD PTP P152 CONT Vel=100 % PDAT161 Tool[1]:GUN X1 Base[2]:Accelo;%{PE}%R 8.2.20,%MKUKATPBASIS,%CMOVE,%VPTP,%P 1:PTP, 2:P152, 3:C_DIS, 5:100, 7:PDAT161
$BWDSTART=FALSE
PDAT_ACT=PPDAT161
FDAT_ACT=FP152
BAS(#PTP_PARAMS,100)
PTP XP152 C_DIS
;ENDFOLD
;FOLD PTP P141 CONT Vel=100 % PDAT147 Tool[1]:GUN X1 Base[2]:Accelo;%{PE}%R 8.2.20,%MKUKATPBASIS,%CMOVE,%VPTP,%P 1:PTP, 2:P141, 3:C_DIS, 5:100, 7:PDAT147
$BWDSTART=FALSE
PDAT_ACT=PPDAT147
FDAT_ACT=FP141
BAS(#PTP_PARAMS,100)
PTP XP141 C_DIS
;ENDFOLD
;FOLD PTP lx610 CONT Vel=100 % P_OLP90 Tool[1]:GUN X1 Base[2]:Accelo;%{PE}%R 8.2.20,%MKUKATPBASIS,%CMOVE,%VPTP,%P 1:PTP, 2:lx610, 3:C_DIS, 5:100, 7:P_OLP90
$BWDSTART=FALSE
PDAT_ACT=PP_OLP90
FDAT_ACT=Flx610
BAS(#PTP_PARAMS,100)
PTP Xlx610 C_DIS
;ENDFOLD
;FOLD PTP P142 CONT Vel=100 % PDAT148 Tool[1]:GUN X1 Base[2]:Accelo;%{PE}%R 8.2.20,%MKUKATPBASIS,%CMOVE,%VPTP,%P 1:PTP, 2:P142, 3:C_DIS, 5:100, 7:PDAT148
$BWDSTART=FALSE
PDAT_ACT=PPDAT148
FDAT_ACT=FP142
BAS(#PTP_PARAMS,100)
PTP XP142 C_DIS
;ENDFOLD

;FOLD OUT 3348 'Fora area GEOBOX' State=TRUE ;%{PE}%R 8.2.20,%MKUKATPBASIS,%COUT,%VOUTX,%P 2:3348, 3:Fora area GEOBOX, 5:TRUE, 6:
$OUT[3348]=TRUE
;ENDFOLD

END

--- ps_ltc_geo_x1.dat ---
&ACCESS RVO2
&REL 17
&COMMENT Solda GUN X1 geometria
&PARAM DISKPATH = KRC:\R1\Program\SOLDA LTC
DEFDAT  ps_ltc_geo_x1
;FOLD EXTERNAL DECLARATIONS;%{PE}%MKUKATPBASIS,%CEXT,%VCOMMON,%P
;FOLD GRIPPERTECH EXT
EXT  H50 (INT  :IN,INT  :IN,INT  :IN,GRP_TYP  :IN )
;ENDFOLD (GRIPPERTECH EXT)
;FOLD SPOTTECH EXT
EXT  USERSPOT (S_COMMAND  :IN,SPOT_TYPE  :IN )
;ENDFOLD (SPOTTECH EXT)
;FOLD BASISTECH EXT;%{PE}%MKUKATPBASIS,%CEXT,%VEXT,%P
EXT  BAS (BAS_COMMAND  :IN,REAL  :IN )
DECL INT SUCCESS
;ENDFOLD (BASISTECH EXT)
;FOLD USER EXT;%{E}%MKUKATPUSER,%CEXT,%VEXT,%P
;Make your modifications here

;ENDFOLD (USER EXT)
;ENDFOLD (EXTERNAL DECLARATIONS)

;# ============ START PATH : swp_p13050r1_ltc_geo_x1 =============
DECL FDAT Fswp_60_0263={TOOL_NO 1,BASE_NO 2,IPO_FRAME #BASE,POINT2[] " "}
DECL SPOT_TYPE SS_OLP1={GUN 1,PAIR #FIRST,RETR #OPN,CLO_TM 0,PGNO1 1,PRESS1 1.0,PGNO2 0,PRESS2 0.0}
DECL E6POS Xswp_60_0263={X -275.645294,Y -980.43219,Z -166.443405,A 34.8704796,B 19.2542801,C 18.5798302,S 2,T 34,E1 -5647.1792,E2 0.0,E3 0.0,E4 0.0,E5 0.0,E6 0.0}
DECL FDAT Fswp_60_0267={TOOL_NO 1,BASE_NO 2,IPO_FRAME #BASE,POINT2[] " "}
DECL SPOT_TYPE SS_OLP2={GUN 1,PAIR #FIRST,RETR #OPN,CLO_TM 0,PGNO1 1,PRESS1 1.0,PGNO2 0,PRESS2 0.0}
DECL E6POS Xswp_60_0267={X -213.047607,Y -1048.96594,Z -164.542007,A 29.3044491,B 19.3898506,C 1.51828504,S 2,T 34,E1 -5647.19092,E2 0.0,E3 0.0,E4 0.0,E5 0.0,E6 0.0}
DECL FDAT Fswp_60_0283={TOOL_NO 1,BASE_NO 2,IPO_FRAME #BASE,POINT2[] " ",TQ_STATE FALSE}
DECL SPOT_TYPE SS_OLP3={GUN 1,PAIR #FIRST,RETR #OPN,CLO_TM 0,PGNO1 1,PRESS1 1.0,PGNO2 0,PRESS2 0.0}
DECL E6POS Xswp_60_0283={X 6.83988285,Y -1239.21399,Z 8.94310188,A 56.0263596,B 24.5332108,C -20.6315804,S 2,T 2,E1 -5181.69385,E2 0.0,E3 0.0,E4 0.0,E5 0.0,E6 0.0}
DECL SPOT_TYPE SS_OLP4={GUN 1,PAIR #FIRST,RETR #OPN,CLO_TM 0,PGNO1 1,PRESS1 1.0,PGNO2 0,PRESS2 0.0}
DECL SPOT_TYPE SS_OLP5={GUN 1,PAIR #FIRST,RETR #OPN,CLO_TM 0,PGNO1 1,PRESS1 1.0,PGNO2 0,PRESS2 0.0}
DECL FDAT Fswp_60_0349={TOOL_NO 1,BASE_NO 2,IPO_FRAME #BASE,POINT2[] " "}
DECL SPOT_TYPE SS_OLP6={GUN 1,PAIR #FIRST,RETR #OPN,CLO_TM 0,PGNO1 1,PRESS1 1.0,PGNO2 0,PRESS2 0.0}
DECL E6POS Xswp_60_0349={X 432.562195,Y -1705.31201,Z 116.379097,A 40.3507309,B 4.63222885,C -89.5844727,S 2,T 2,E1 -4540.75293,E2 0.0,E3 0.0,E4 0.0,E5 0.0,E6 0.0}
DECL FDAT Fswp_60_0355={TOOL_NO 1,BASE_NO 2,IPO_FRAME #BASE,POINT2[] " "}
DECL SPOT_TYPE SS_OLP7={GUN 1,PAIR #FIRST,RETR #OPN,CLO_TM 0,PGNO1 1,PRESS1 1.0,PGNO2 0,PRESS2 0.0}
DECL E6POS Xswp_60_0355={X 421.169403,Y -1718.13696,Z 279.697906,A 40.9335289,B -3.80524111,C -88.8869324,S 2,T 2,E1 -4540.78711,E2 0.0,E3 0.0,E4 0.0,E5 0.0,E6 0.0}
DECL FDAT Fswp_60_0317={TOOL_NO 1,BASE_NO 2,IPO_FRAME #BASE,POINT2[] " "}
DECL SPOT_TYPE SS_OLP8={GUN 1,PAIR #FIRST,RETR #OPN,CLO_TM 0,PGNO1 1,PRESS1 1.0,PGNO2 0,PRESS2 0.0}
DECL E6POS Xswp_60_0317={X 308.307007,Y -1610.21399,Z 6.46468401,A 127.521103,B -4.08989096,C 144.1259,S 2,T 10,E1 -4568.79297,E2 0.0,E3 0.0,E4 0.0,E5 0.0,E6 0.0}
DECL FDAT Fswp_60_0321={TOOL_NO 1,BASE_NO 2,IPO_FRAME #BASE,POINT2[] " ",TQ_STATE FALSE}
DECL SPOT_TYPE SS_OLP9={GUN 1,PAIR #FIRST,RETR #OPN,CLO_TM 0,PGNO1 1,PRESS1 1.0,PGNO2 0,PRESS2 0.0}
DECL E6POS Xswp_60_0321={X 337.849487,Y -1672.93506,Z -9.62210846,A 128.600006,B 1.93651104,C 143.567093,S 2,T 10,E1 -4568.6748,E2 0.0,E3 0.0,E4 0.0,E5 0.0,E6 0.0}
DECL FDAT Fswp_60_0325={TOOL_NO 1,BASE_NO 2,IPO_FRAME #BASE,POINT2[] " ",TQ_STATE FALSE}
DECL SPOT_TYPE SS_OLP10={GUN 1,PAIR #FIRST,RETR #OPN,CLO_TM 0,PGNO1 1,PRESS1 1.0,PGNO2 0,PRESS2 0.0}
DECL E6POS Xswp_60_0325={X 397.010406,Y -1691.29297,Z 3.9759531,A 119.003899,B -5.36455393,C 137.756195,S 2,T 10,E1 -4568.69678,E2 0.0,E3 0.0,E4 0.0,E5 0.0,E6 0.0}
DECL BASIS_SUGG_T LAST_BASIS={POINT1[] "PS01010001              ",POINT2[] "PS01010001              ",CP_PARAMS[] "CPDAT0                  ",PTP_PARAMS[] "PDAT0                   ",CONT[] "                        ",CP_VEL[] "2.0                     ",PTP_VEL[] " 100                    ",SPL_NAME[] "S0                      "}
DECL SPOT_SUGG_T LAST_SPOT={GUN[] "4                       ",RETR_CMD[] "#CLO                    ",CHOISE[] "#FIRST                  ",CLO_TM[] "1                       ",PGNO1[] "189                     ",PRESS1[] "0                       ",PGNO2[] "1                       ",PRESS2[] "0                       ",SPOT_PARAMS[] "NORMAL                  "}
DECL E6POS Xswp_60_0327={X -1825.44104,Y -6414.63623,Z 1659.75806,A -116.622902,B -6.43793201,C 136.093307,S 2,T 10,E1 -4568.69678,E2 0.0,E3 0.0,E4 0.0,E5 0.0,E6 0.0}
DECL FDAT Fswp_60_0327={TOOL_NO 1,BASE_NO 0,IPO_FRAME #BASE,POINT2[] " ",TQ_STATE FALSE}
DECL E6POS XP63={X 149.8685,Y -2567.51904,Z -128.437103,A 141.404694,B 27.8619308,C 99.6784897,S 2,T 10,E1 -4460.36279,E2 0.0,E3 0.0,E4 0.0,E5 0.0,E6 0.0}
DECL FDAT FP63={TOOL_NO 1,BASE_NO 2,IPO_FRAME #BASE,POINT2[] " ",TQ_STATE FALSE}
DECL PDAT PPDAT65={VEL 100.0,ACC 100.0,APO_DIST 100.0,APO_MODE #CDIS}
DECL E6POS XP112={X 128.800003,Y -2931.58496,Z -129.202301,A 55.0395699,B 45.2179985,C -42.0333595,S 2,T 2,E1 -3987.91797,E2 0.0,E3 0.0,E4 0.0,E5 0.0,E6 0.0}
DECL FDAT FP112={TOOL_NO 1,BASE_NO 2,IPO_FRAME #BASE,POINT2[] " ",TQ_STATE FALSE}
DECL PDAT PPDAT114={VEL 100.0,ACC 100.0,APO_DIST 100.0,APO_MODE #CDIS}
DECL PDAT PPDAT115={VEL 100.0,ACC 100.0,APO_DIST 100.0,APO_MODE #CDIS}
DECL E6POS XP113={X 223.016495,Y -1989.22095,Z 257.250488,A 40.7202988,B 3.102386,C -89.7601089,S 2,T 2,E1 -4540.78809,E2 0.0,E3 0.0,E4 0.0,E5 0.0,E6 0.0}
DECL FDAT FP113={TOOL_NO 1,BASE_NO 2,IPO_FRAME #BASE,POINT2[] " ",TQ_STATE FALSE}
DECL PDAT PPDAT116={VEL 100.0,ACC 100.0,APO_DIST 100.0,APO_MODE #CDIS}
DECL E6POS XP114={X 445.128204,Y -1749.01599,Z 250.443405,A 40.6904488,B -7.20178699,C -88.9869919,S 2,T 2,E1 -4540.78809,E2 0.0,E3 0.0,E4 0.0,E5 0.0,E6 0.0}
DECL FDAT FP114={TOOL_NO 1,BASE_NO 2,IPO_FRAME #BASE,POINT2[] " ",TQ_STATE FALSE}
DECL PDAT PP_OLP80={VEL 100.0,ACC 100.0,APO_DIST 0.0}
DECL PDAT PP_OLP81={VEL 100.0,ACC 100.0,APO_DIST 0.0}
DECL PDAT PPDAT117={VEL 100.0,ACC 100.0,APO_DIST 100.0,APO_MODE #CDIS}
DECL E6POS XP115={X 465.378387,Y -1730.63098,Z 102.938698,A 41.4731293,B 6.24935913,C -89.4617996,S 2,T 2,E1 -4540.75293,E2 0.0,E3 0.0,E4 0.0,E5 0.0,E6 0.0}
DECL FDAT FP115={TOOL_NO 1,BASE_NO 2,IPO_FRAME #BASE,POINT2[] " ",TQ_STATE FALSE}
DECL PDAT PP_OLP82={VEL 100.0,ACC 100.0,APO_DIST 100.0,APO_MODE #CDIS}
DECL E6POS Xlx695={X 247.467102,Y -1983.28699,Z 117.566002,A 40.3175316,B 0.397013813,C -89.5861206,S 2,T 2,E1 -4540.75293,E2 0.0,E3 0.0,E4 0.0,E5 0.0,E6 0.0}
DECL FDAT Flx695={TOOL_NO 1,BASE_NO 2,IPO_FRAME #BASE,POINT2[] " "}
DECL PDAT PPDAT119={VEL 100.0,ACC 100.0,APO_DIST 100.0,APO_MODE #CDIS}
DECL E6POS XP117={X -805.128296,Y -1482.06897,Z -24.73699,A 47.0636597,B 2.3741219,C -3.5756309,S 2,T 34,E1 -5647.1958,E2 0.0,E3 0.0,E4 0.0,E5 0.0,E6 0.0}
DECL FDAT FP117={TOOL_NO 1,BASE_NO 2,IPO_FRAME #BASE,POINT2[] " ",TQ_STATE FALSE}
DECL PDAT PPDAT120={VEL 100.0,ACC 100.0,APO_DIST 100.0,APO_MODE #CDIS}
DECL E6POS XP118={X -501.282806,Y -1183.51904,Z -151.957703,A 31.5826492,B 14.4653196,C -0.0970954373,S 2,T 34,E1 -5647.20117,E2 0.0,E3 0.0,E4 0.0,E5 0.0,E6 0.0}
DECL FDAT FP118={TOOL_NO 1,BASE_NO 2,IPO_FRAME #BASE,POINT2[] " ",TQ_STATE FALSE}
DECL PDAT PPDAT121={VEL 100.0,ACC 100.0,APO_DIST 100.0,APO_MODE #CDIS}
DECL PDAT PPDAT122={VEL 100.0,ACC 100.0,APO_DIST 100.0,APO_MODE #CDIS}
DECL E6POS XP120={X -240.307999,Y -1027.03699,Z -175.615204,A 32.5320892,B 19.41992,C 4.54465485,S 2,T 34,E1 -5647.1748,E2 0.0,E3 0.0,E4 0.0,E5 0.0,E6 0.0}
DECL FDAT FP120={TOOL_NO 1,BASE_NO 2,IPO_FRAME #BASE,POINT2[] " ",TQ_STATE FALSE}
DECL PDAT PPDAT123={VEL 100.0,ACC 100.0,APO_DIST 100.0,APO_MODE #CDIS}
DECL PDAT PP_OLP83={VEL 100.0,ACC 100.0,APO_DIST 100.0,APO_MODE #CDIS}
DECL E6POS Xlx696={X -459.795898,Y -1097.73706,Z -165.608002,A 36.6101303,B 19.1170197,C 8.19668961,S 2,T 34,E1 -5647.1748,E2 0.0,E3 0.0,E4 0.0,E5 0.0,E6 0.0}
DECL FDAT Flx696={TOOL_NO 1,BASE_NO 2,IPO_FRAME #BASE,POINT2[] " "}
DECL PDAT PP_OLP84={VEL 100.0,ACC 100.0,APO_DIST 100.0,APO_MODE #CDIS}
DECL E6POS Xlx697={X -805.127625,Y -1482.06995,Z -24.7408199,A 47.0636292,B 2.37426209,C -3.57572389,S 2,T 34,E1 -5647.1958,E2 0.0,E3 0.0,E4 0.0,E5 0.0,E6 0.0}
DECL FDAT Flx697={TOOL_NO 1,BASE_NO 2,IPO_FRAME #BASE,POINT2[] " "}
DECL PDAT PPDAT124={VEL 100.0,ACC 100.0,APO_DIST 80.0,APO_MODE #CDIS}
DECL E6POS XP122={X -339.747314,Y -1530.125,Z 57.2784996,A 62.6198311,B 11.3163099,C -12.12533,S 2,T 34,E1 -5181.66406,E2 0.0,E3 0.0,E4 0.0,E5 0.0,E6 0.0}
DECL FDAT FP122={TOOL_NO 1,BASE_NO 2,IPO_FRAME #BASE,POINT2[] " ",TQ_STATE FALSE}
DECL PDAT PPDAT125={VEL 100.0,ACC 50.0,APO_DIST 80.0,APO_MODE #CDIS}
DECL E6POS XP123={X -119.906601,Y -1419.73999,Z 23.3350296,A 66.8781586,B 12.7666798,C -15.6264,S 2,T 34,E1 -5181.68896,E2 0.0,E3 0.0,E4 0.0,E5 0.0,E6 0.0}
DECL FDAT FP123={TOOL_NO 1,BASE_NO 2,IPO_FRAME #BASE,POINT2[] " ",TQ_STATE FALSE}
DECL PDAT PPDAT126={VEL 100.0,ACC 50.0,APO_DIST 50.0,APO_MODE #CDIS}
DECL E6POS XP124={X -47.9475403,Y -1344.42505,Z 30.1196709,A 61.2519112,B 11.1653605,C -16.7942009,S 2,T 34,E1 -5181.68896,E2 0.0,E3 0.0,E4 0.0,E5 0.0,E6 0.0}
DECL FDAT FP124={TOOL_NO 1,BASE_NO 2,IPO_FRAME #BASE,POINT2[] " ",TQ_STATE FALSE}
DECL PDAT PPDAT127={VEL 100.0,ACC 50.0,APO_DIST 10.0,APO_MODE #CDIS}
DECL E6POS XP125={X -13.6633902,Y -1303.02698,Z 7.46283007,A 59.4785385,B 22.2280293,C -12.3178396,S 2,T 2,E1 -5181.68994,E2 0.0,E3 0.0,E4 0.0,E5 0.0,E6 0.0}
DECL FDAT FP125={TOOL_NO 1,BASE_NO 2,IPO_FRAME #BASE,POINT2[] " ",TQ_STATE FALSE}
DECL PDAT PP_OLP85={VEL 100.0,ACC 100.0,APO_DIST 0.0}
DECL PDAT PPDAT128={VEL 100.0,ACC 100.0,APO_DIST 15.0,APO_MODE #CDIS}
DECL E6POS XP126={X -48.0881805,Y -1344.44995,Z 26.9599705,A 59.0536118,B 21.2694607,C -19.8021393,S 2,T 2,E1 -5181.69092,E2 0.0,E3 0.0,E4 0.0,E5 0.0,E6 0.0}
DECL FDAT FP126={TOOL_NO 1,BASE_NO 2,IPO_FRAME #BASE,POINT2[] " ",TQ_STATE FALSE}
DECL PDAT PPDAT129={VEL 100.0,ACC 100.0,APO_DIST 20.0,APO_MODE #CDIS}
DECL E6POS XP127={X -141.712997,Y -1441.54504,Z 32.7751389,A 65.8396912,B 14.4452696,C -20.0396709,S 2,T 34,E1 -5181.68896,E2 0.0,E3 0.0,E4 0.0,E5 0.0,E6 0.0}
DECL FDAT FP127={TOOL_NO 1,BASE_NO 2,IPO_FRAME #BASE,POINT2[] " ",TQ_STATE FALSE}
DECL PDAT PPDAT134={VEL 100.0,ACC 100.0,APO_DIST 30.0,APO_MODE #CDIS}
DECL E6POS XP132={X -103.123703,Y -1698.18103,Z 59.301899,A 62.4764595,B 22.6058006,C -7.61601782,S 2,T 2,E1 -5181.7041,E2 0.0,E3 0.0,E4 0.0,E5 0.0,E6 0.0}
DECL FDAT FP132={TOOL_NO 1,BASE_NO 2,IPO_FRAME #BASE,POINT2[] " ",TQ_STATE FALSE}
DECL E6POS XP134={X 375.866486,Y -2553.52197,Z 94.818222,A 62.3175812,B 37.8605804,C -34.3857384,S 2,T 2,E1 -4175.70215,E2 0.0,E3 0.0,E4 0.0,E5 0.0,E6 0.0}
DECL FDAT FP134={TOOL_NO 1,BASE_NO 2,IPO_FRAME #BASE,POINT2[] " ",TQ_STATE FALSE}
DECL PDAT PPDAT136={VEL 100.0,ACC 100.0,APO_DIST 50.0,APO_MODE #CDIS}
DECL E6POS XP135={X 219.481094,Y -2785.84912,Z -130.159302,A 126.799698,B 53.5773201,C 39.0210495,S 2,T 10,E1 -4184.32813,E2 0.0,E3 0.0,E4 0.0,E5 0.0,E6 0.0}
DECL FDAT FP135={TOOL_NO 1,BASE_NO 2,IPO_FRAME #BASE,POINT2[] " ",TQ_STATE FALSE}
DECL PDAT PPDAT137={VEL 100.0,ACC 100.0,APO_DIST 100.0,APO_MODE #CDIS}
DECL PDAT PPDAT138={VEL 100.0,ACC 100.0,APO_DIST 100.0,APO_MODE #CDIS}
DECL E6POS XP136={X 429.565491,Y -1841.61304,Z -4.86375713,A 129.667999,B -2.37908912,C 148.920502,S 2,T 10,E1 -4568.75293,E2 0.0,E3 0.0,E4 0.0,E5 0.0,E6 0.0}
DECL FDAT FP136={TOOL_NO 1,BASE_NO 2,IPO_FRAME #BASE,POINT2[] " ",TQ_STATE FALSE}
DECL PDAT PP_OLP88={VEL 100.0,ACC 100.0,APO_DIST 100.0,APO_MODE #CDIS}
DECL E6POS Xlx698={X 292.525299,Y -1643.73096,Z -4.86532784,A 129.667999,B -2.37911105,C 148.920502,S 2,T 10,E1 -4568.75293,E2 0.0,E3 0.0,E4 0.0,E5 0.0,E6 0.0}
DECL FDAT Flx698={TOOL_NO 1,BASE_NO 2,IPO_FRAME #BASE,POINT2[] " "}
DECL PDAT PP_OLP89={VEL 100.0,ACC 100.0,APO_DIST 0.0}
DECL PDAT PPDAT139={VEL 100.0,ACC 100.0,APO_DIST 100.0,APO_MODE #CDIS}
DECL PDAT PPDAT140={VEL 100.0,ACC 100.0,APO_DIST 100.0,APO_MODE #CDIS}
DECL PDAT PPDAT141={VEL 100.0,ACC 100.0,APO_DIST 100.0,APO_MODE #CDIS}
DECL PDAT PPDAT146={VEL 100.0,ACC 100.0,APO_DIST 100.0,APO_MODE #CDIS}
DECL E6POS XP140={X 501.628906,Y -1918.77502,Z -26.8826199,A 116.119301,B 3.38413692,C 148.564102,S 2,T 10,E1 -4460.36279,E2 0.0,E3 0.0,E4 0.0,E5 0.0,E6 0.0}
DECL FDAT FP140={TOOL_NO 1,BASE_NO 2,IPO_FRAME #BASE,POINT2[] " ",TQ_STATE FALSE}
DECL PDAT PPDAT147={VEL 100.0,ACC 100.0,APO_DIST 100.0,APO_MODE #CDIS}
DECL E6POS XP141={X 149.8685,Y -2567.51904,Z -128.437103,A 141.404694,B 27.8619308,C 99.6784897,S 2,T 10,E1 -4460.36279,E2 0.0,E3 0.0,E4 0.0,E5 0.0,E6 0.0}
DECL FDAT FP141={TOOL_NO 1,BASE_NO 2,IPO_FRAME #BASE,POINT2[] " ",TQ_STATE FALSE}
DECL PDAT PP_OLP90={VEL 100.0,ACC 100.0,APO_DIST 100.0,APO_MODE #CDIS}
DECL E6POS Xlx610={X 192.240097,Y -2890.06006,Z -302.896515,A 132.393799,B 56.4223709,C 43.6062698,S 2,T 10,E1 -4184.32715,E2 0.0,E3 0.0,E4 0.0,E5 0.0,E6 0.0}
DECL FDAT Flx610={TOOL_NO 1,BASE_NO 2,IPO_FRAME #BASE,POINT2[] " "}
DECL PDAT PPDAT148={VEL 100.0,ACC 100.0,APO_DIST 100.0,APO_MODE #CDIS}
DECL E6POS XP142={X -20.6214809,Y -2868.67896,Z 427.8992,A 112.6278,B 26.7825699,C -22.8124199,S 2,T 2,E1 -3881.30811,E2 0.0,E3 0.0,E4 0.0,E5 0.0,E6 0.0}
DECL FDAT FP142={TOOL_NO 1,BASE_NO 2,IPO_FRAME #BASE,POINT2[] " ",TQ_STATE FALSE}
DECL PDAT PPDAT149={VEL 100.0,ACC 100.0,APO_DIST 100.0,APO_MODE #CDIS}
DECL E6POS XP143={X 301.243286,Y -1617.51001,Z 20.1037693,A 125.285301,B -8.34358597,C 149.555496,S 2,T 10,E1 -4568.78613,E2 0.0,E3 0.0,E4 0.0,E5 0.0,E6 0.0}
DECL FDAT FP143={TOOL_NO 1,BASE_NO 2,IPO_FRAME #BASE,POINT2[] " ",TQ_STATE FALSE}
DECL PDAT PPDAT150={VEL 100.0,ACC 100.0,APO_DIST 100.0,APO_MODE #CDIS}
DECL E6POS XP144={X 301.243286,Y -1617.51001,Z 20.1037693,A 125.285301,B -8.34358597,C 149.555496,S 2,T 10,E1 -4568.78613,E2 0.0,E3 0.0,E4 0.0,E5 0.0,E6 0.0}
DECL FDAT FP144={TOOL_NO 1,BASE_NO 2,IPO_FRAME #BASE,POINT2[] " ",TQ_STATE FALSE}
DECL PDAT PPDAT151={VEL 100.0,ACC 100.0,APO_DIST 100.0,APO_MODE #CDIS}
DECL E6POS Xswp_60_0315={X -1817.73596,Y -6538.56104,Z 1664.00903,A -105.512199,B -11.0989103,C 149.779205,S 2,T 10,E1 -4568.79785,E2 0.0,E3 0.0,E4 0.0,E5 0.0,E6 0.0}
DECL FDAT Fswp_60_0315={TOOL_NO 1,BASE_NO 0,IPO_FRAME #BASE,POINT2[] " ",TQ_STATE FALSE}
DECL E6POS XP145={X 291.662994,Y -1617.43896,Z -5.96740818,A 127.521301,B -4.09028482,C 144.125793,S 2,T 10,E1 -4568.79297,E2 0.0,E3 0.0,E4 0.0,E5 0.0,E6 0.0}
DECL FDAT FP145={TOOL_NO 1,BASE_NO 2,IPO_FRAME #BASE,POINT2[] " ",TQ_STATE FALSE}
DECL PDAT PPDAT152={VEL 100.0,ACC 100.0,APO_DIST 100.0,APO_MODE #CDIS}
DECL E6POS XP146={X 402.0242,Y -1685.71204,Z 23.6734409,A 111.884201,B -6.74503803,C 137.101501,S 2,T 10,E1 -4568.69678,E2 0.0,E3 0.0,E4 0.0,E5 0.0,E6 0.0}
DECL FDAT FP146={TOOL_NO 1,BASE_NO 2,IPO_FRAME #BASE,POINT2[] " ",TQ_STATE FALSE}
DECL PDAT PPDAT153={VEL 100.0,ACC 100.0,APO_DIST 100.0,APO_MODE #CDIS}
DECL E6POS XP147={X -11.8331299,Y -1323.75098,Z 0.671140611,A 58.5486107,B 17.0795193,C -15.2183399,S 2,T 34,E1 -5181.69092,E2 0.0,E3 0.0,E4 0.0,E5 0.0,E6 0.0}
DECL FDAT FP147={TOOL_NO 1,BASE_NO 2,IPO_FRAME #BASE,POINT2[] " ",TQ_STATE FALSE}
DECL PDAT PPDAT154={VEL 100.0,ACC 100.0,APO_DIST 80.0,APO_MODE #CDIS}
DECL PDAT PPDAT155={VEL 100.0,ACC 100.0,APO_DIST 100.0,APO_MODE #CDIS}
DECL E6POS Xswp_60_0331={X 319.516693,Y -1653.85706,Z -10.5840397,A 125.3731,B -3.16019797,C 145.238007,S 2,T 10,E1 -4568.69287,E2 0.0,E3 0.0,E4 0.0,E5 0.0,E6 0.0}
DECL FDAT Fswp_60_0331={TOOL_NO 1,BASE_NO 2,IPO_FRAME #BASE,POINT2[] " ",TQ_STATE FALSE}
DECL PDAT PPDAT156={VEL 100.0,ACC 100.0,APO_DIST 100.0,APO_MODE #CDIS}
DECL E6POS Xswp_60_0332={X 357.036591,Y -1691.21399,Z -9.36073685,A 128.599792,B 1.937621,C 143.567398,S 2,T 10,E1 -4568.6748,E2 0.0,E3 0.0,E4 0.0,E5 0.0,E6 0.0}
DECL FDAT Fswp_60_0332={TOOL_NO 1,BASE_NO 2,IPO_FRAME #BASE,POINT2[] " ",TQ_STATE FALSE}
DECL E6POS XP148={X 375.404388,Y -1714.22498,Z -8.3659811,A 128.599792,B 1.93763995,C 143.567505,S 2,T 10,E1 -4568.6748,E2 0.0,E3 0.0,E4 0.0,E5 0.0,E6 0.0}
DECL FDAT FP148={TOOL_NO 1,BASE_NO 2,IPO_FRAME #BASE,POINT2[] " ",TQ_STATE FALSE}
DECL PDAT PPDAT157={VEL 100.0,ACC 100.0,APO_DIST 80.0,APO_MODE #CDIS}
DECL E6POS XP149={X 387.077789,Y -1711.75806,Z 4.77827501,A 123.195396,B -3.82490492,C 140.115799,S 2,T 10,E1 -4568.68896,E2 0.0,E3 0.0,E4 0.0,E5 0.0,E6 0.0}
DECL FDAT FP149={TOOL_NO 1,BASE_NO 2,IPO_FRAME #BASE,POINT2[] " ",TQ_STATE FALSE}
DECL PDAT PPDAT158={VEL 100.0,ACC 100.0,APO_DIST 80.0,APO_MODE #CDIS}
DECL E6POS XP150={X 375.227386,Y -1691.30896,Z 21.6169395,A 116.706001,B -6.07782602,C 141.961105,S 2,T 10,E1 -4558.85889,E2 0.0,E3 0.0,E4 0.0,E5 0.0,E6 0.0}
DECL FDAT FP150={TOOL_NO 1,BASE_NO 2,IPO_FRAME #BASE,POINT2[] " ",TQ_STATE FALSE}
DECL PDAT PPDAT159={VEL 100.0,ACC 100.0,APO_DIST 100.0,APO_MODE #CDIS}
DECL E6POS XP151={X 355.217285,Y -1727.13794,Z 9.44879627,A 123.858902,B 0.442456514,C 146.9021,S 2,T 10,E1 -4533.8042,E2 0.0,E3 0.0,E4 0.0,E5 0.0,E6 0.0}
DECL FDAT FP151={TOOL_NO 1,BASE_NO 2,IPO_FRAME #BASE,POINT2[] " ",TQ_STATE FALSE}
DECL PDAT PPDAT160={VEL 100.0,ACC 100.0,APO_DIST 100.0,APO_MODE #CDIS}
DECL E6POS XP152={X 532.498291,Y -2000.23901,Z 8.68222904,A 118.759499,B 5.11184788,C 130.077805,S 2,T 10,E1 -4460.36279,E2 0.0,E3 0.0,E4 0.0,E5 0.0,E6 0.0}
DECL FDAT FP152={TOOL_NO 1,BASE_NO 2,IPO_FRAME #BASE,POINT2[] " ",TQ_STATE FALSE}
DECL PDAT PPDAT161={VEL 100.0,ACC 100.0,APO_DIST 100.0,APO_MODE #CDIS}
ENDDAT
